{attribute 'linkalways'} 
{attribute 'no_explicit_call' := 'This FB is a CLASS and must be accessed using methods or properties'}
{attribute 'enable_dynamic_creation'}
FUNCTION_BLOCK FINAL MUL_DWORD EXTENDS Node
VAR
	in1 : _DWORD(0);
	in2 : _DWORD(0);
	out : _DWORD(0);
END_VAR

METHOD PUBLIC Clone : I_Node
VAR
	pNode : POINTER TO MUL_DWORD;
END_VAR
pNode := __NEW(MUL_DWORD);
Clone := pNode^;
END_METHOD

METHOD FB_init : BOOL
VAR_INPUT
	bInitRetains : BOOL; // if TRUE, the retain variables are initialized (warm start / cold start)
	bInCopyCode : BOOL;  // if TRUE, the instance afterwards gets moved into the copy code (online change)
END_VAR
AddInput('in1',THIS^.in1);
AddInput('in2',THIS^.in2);
AddOutput('out', THIS^.out);
END_METHOD

METHOD PROTECTED OnExecute
VAR
END_VAR
out.Value := in1.Value * in2.Value;
END_METHOD

END_FUNCTION_BLOCK

(* stored: Version 1.1.0.1, ProductVersion 3.1.4024.15
   POU MUL_DWORD: Id {7429dc09-14f6-4053-8aaa-8f00b695f294}, SpecialFunc None
   Folder Constructor: Id {8c070adf-a572-46e5-9679-a23e40fde630}
   Method Clone: Id {eef091c9-d5a7-4edb-b308-1b5d654bbd2e}
   Method FB_init: Id {c8c7a0c7-6408-4c7b-8315-cd60cdf03ceb}
   Method OnExecute: Id {7cdb2885-4d67-4d53-8341-1eeaa06fb738} *)
